Fanuc KAREL source: kf00079.KL

-- PROVISIONAL review KL for V940-1; original PC SHA256 45a5c7874d5fe9aabf29384aed1f4ce66012bbbbf487ff4fee3a9a0870246dba
-- Incomplete behavior may be omitted. Consult companion uncertainty JSON. Do not deploy.
PROGRAM KF00079
%NOLOCKGROUP
BEGIN
  -- V9_ZERO_TABLE_METADATA_HINT layout=0002_ascii; no indexed target words; source/name/runtime held
  -- UNRESOLVED_PC offsets 5-15; opcodes 3F,75
  -- UNRESOLVED_PC offsets 20-29; opcodes 3F,75
  -- UNRESOLVED_PC offsets 34-45; opcodes 2E,23
  -- UNRESOLVED_PC offsets 50-61; opcodes 2E,23
  -- UNRESOLVED_PC offsets 66-84; opcodes 27,22,2A,22,31
  -- UNRESOLVED_PC offsets 89-93; opcodes 7F
END KF00079
